// Valve control logic (fill by default, discharge if TargetWaterLevel and CurrentWaterLevel are swapped)
FUNCTION_BLOCK PUBLIC ValveController
VAR_INPUT
	TargetWaterLevel: REAL;
	CurrentWaterLevel: REAL;
	// The value (cm) at which the flow speed will start to decrease linearly
	ScaleMax : INT;
END_VAR
VAR_OUTPUT
	AnalogOutputValue: WORD;
END_VAR
VAR
	LevelOffset : REAL;
	AnalogOutputTemp: WORD;
END_VAR

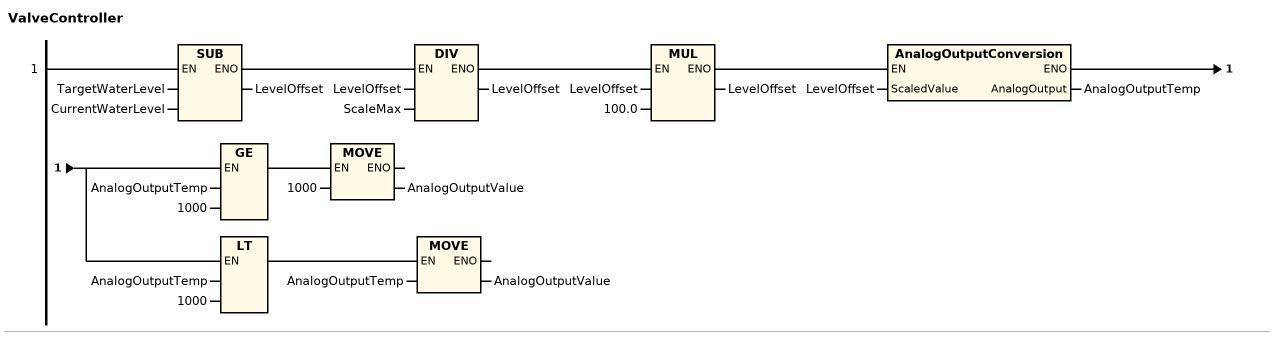
// NETWORK 1
LevelOffset := TargetWaterLevel - CurrentWaterLevel;
LevelOffset := LevelOffset / ScaleMax;
LevelOffset := LevelOffset * 100.0;
AnalogOutputConversion(ScaledValue := LevelOffset, AnalogOutput => AnalogOutputTemp);
IF AnalogOutputTemp >= 1000 THEN AnalogOutputValue := 1000; END_IF
IF AnalogOutputTemp < 1000 THEN AnalogOutputValue := AnalogOutputTemp; END_IF

END_FUNCTION_BLOCK

(* stored: Version 1.1.0.1, ProductVersion 3.1.4024.12
   POU ValveController: Id {45f1b5a4-0773-41c0-bb1b-65f0fb403878}, SpecialFunc None *)
